# EPICS substitutions: epics/db/EL9505.substitutions
file "./db/ecSlave.template"
{
  pattern {}
          {}
}

file "./db/EL9505.template"
{
  pattern {}
          {}
}
